FUNCTION_BLOCK Revezamento_2_Motores (* Composite Function Block Type *)
  (* Standard: 61499-2 *)
  (* Version 0.0, 25/02/2026, template *)
  PACKAGE Hidryco.HidrycoLib;
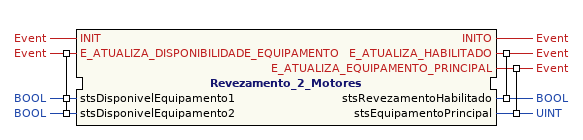
  EVENT_INPUT
    INIT;
    E_ATUALIZA_DISPONIBILIDADE_EQUIPAMENTO WITH stsDisponivelEquipamento1, stsDisponivelEquipamento2;
  END_EVENT
  EVENT_OUTPUT
    INITO;
    E_ATUALIZA_HABILITADO WITH stsRevezamentoHabilitado;
    E_ATUALIZA_EQUIPAMENTO_PRINCIPAL WITH stsEquipamentoPrincipal;
  END_EVENT
  VAR_INPUT
    stsDisponivelEquipamento1 : BOOL;
    stsDisponivelEquipamento2 : BOOL;
  END_VAR
  VAR_OUTPUT
    stsRevezamentoHabilitado : BOOL;
    stsEquipamentoPrincipal : UINT;
  END_VAR
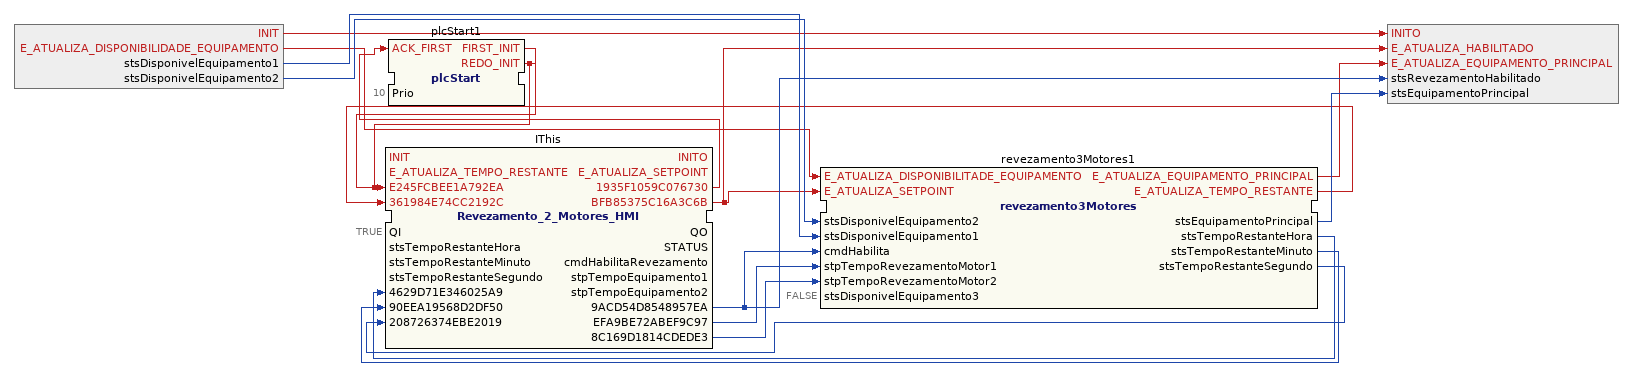
  FBS
    IThis : Revezamento_2_Motores_HMI(QI := TRUE);
    revezamento3Motores1 : revezamento3Motores(stsDisponivelEquipamento3 := FALSE);
    plcStart1 : plcStart(Prio := 10);
  END_FBS
  EVENT_CONNECTIONS
    E_ATUALIZA_DISPONIBILIDADE_EQUIPAMENTO TO revezamento3Motores1.E_ATUALIZA_DISPONIBILITADE_EQUIPAMENTO;
    revezamento3Motores1.E_ATUALIZA_EQUIPAMENTO_PRINCIPAL TO E_ATUALIZA_EQUIPAMENTO_PRINCIPAL;
    plcStart1.FIRST_INIT TO IThis.E245FCBEE1A792EA;
    plcStart1.REDO_INIT TO IThis.E245FCBEE1A792EA;
    revezamento3Motores1.E_ATUALIZA_TEMPO_RESTANTE TO IThis.361984E74CC2192C;
    IThis.1935F1059C076730 TO plcStart1.ACK_FIRST;
    IThis.BFB85375C16A3C6B TO revezamento3Motores1.E_ATUALIZA_SETPOINT;
    IThis.BFB85375C16A3C6B TO E_ATUALIZA_HABILITADO;
    INIT TO INITO;
  END_CONNECTIONS
  DATA_CONNECTIONS
    stsDisponivelEquipamento2 TO revezamento3Motores1.stsDisponivelEquipamento2;
    stsDisponivelEquipamento1 TO revezamento3Motores1.stsDisponivelEquipamento1;
    revezamento3Motores1.stsEquipamentoPrincipal TO stsEquipamentoPrincipal;
    revezamento3Motores1.stsTempoRestanteHora TO IThis.4629D71E346025A9;
    revezamento3Motores1.stsTempoRestanteMinuto TO IThis.90EEA19568D2DF50;
    revezamento3Motores1.stsTempoRestanteSegundo TO IThis.208726374EBE2019;
    IThis.9ACD54D8548957EA TO revezamento3Motores1.cmdHabilita;
    IThis.9ACD54D8548957EA TO stsRevezamentoHabilitado;
    IThis.EFA9BE72ABEF9C97 TO revezamento3Motores1.stpTempoRevezamentoMotor1;
    IThis.8C169D1814CDEDE3 TO revezamento3Motores1.stpTempoRevezamentoMotor2;
  END_CONNECTIONS
END_FUNCTION_BLOCK
